(* PLC project poST.project, poSTIDE *)
(* stored: creationDateTime 2021-08-31T00:00:00.000000 *)

FUNCTION DIV : ANY_NUM
  VAR_INPUT
    in1 : ANY_NUM;
    in2 : ANY_NUM;
  END_VAR

END_FUNCTION
